Staubli VAL3: language.pjx

--- language.pjx ---
Parameters version=s7.2.1 stackSize=5000 millimeterUnit=true
Program file=getLanguage.pgx
Program file=getYesNo.pgx
Program file=message.pgx
Program file=page.pgx
Program file=setLanguage.pgx
Data file=language.dtx
Library alias=language path=Disk://kernel/language/english/english.pjx

--- getLanguage.pgx ---
public program getLanguage(string& x_sPath[])
begin
  x_sPath=language:libPath()
end

--- getYesNo.pgx ---
public program getYesNo(string& x_sYesNo[])
begin
  x_sYesNo=language:Yes
  x_sYesNo[1]=language:No
end

--- message.pgx ---
public program message(string& x_sMessage[], num x_nIndex)
begin
  // load the default one
  call language:message(x_sMessage,x_nIndex)
end

--- page.pgx ---
public program page(string& x_sMenuName[], num x_nIndex)
// set all the page
begin
  // load the default one
  call language:page(x_sMenuName,x_nIndex)
end

--- setLanguage.pgx ---
public program setLanguage(string x_sPath)
  local num l_nResult
  local string l_sMessage
begin
  //
  call language:message(l_sMessage,-7)
  l_nResult=language:libLoad(x_sPath)
  if l_nResult!=0
    popUpMsg(l_sMessage+x_sPath+" ; "+toString("",l_nResult))
  endIf
end
